// TIA Portal V18 export
// export: Created 2026-06-21T12:15:02Z, ExportSetting WithDefaults
PlcWatchTable "WT_PLC2_PID_Sim"
  PlcWatchTableEntry "PID_Bon4_Enable"
  PlcWatchTableEntry "PID_Bon4_SP"
  PlcWatchTableEntry "TT3219_Bon4_Sim"
  PlcWatchTableEntry "TT3219_Bon4_Target"
  PlcWatchTableEntry "PID_Bon4_CV"
  PlcWatchTableEntry "PID_Bon4_Error"
